PROGRAM MAIN
VAR
	machine : Machine;
END_VAR

END_PROGRAM

(* stored: Version 1.1.0.1, ProductVersion 3.1.4024.12
   POU MAIN: Id {3123fd03-aa82-4253-b979-e50f3a78bc29}, SpecialFunc None *)
